                $ 899 "vr2_p3_up≔contact_fun(p[0,0,0,0,0,0],[0,1,0],20000,20,20)"
                global vr2_p3_up=contact_fun(p[0,0,0,0,0,0],[0,1,0],20000,20,20)
                $ 900 "direction(p[0,0,0,0,0,0],[0,-1,0],30,120,160)"
                direction(p[0,0,0,0,0,0],[0,-1,0],30,120,160)
                $ 901 "direction(p[0,0,0,0,0,0],[-1,0,0],20,120,160)"
                direction(p[0,0,0,0,0,0],[-1,0,0],20,120,160)
              end
              $ 902 "A_Touch_p[A_sel_v+9]=touch_4point(vr2_p1_up,vr2_p2_up,vr2_p3_up)"
              A_Touch_p[A_sel_v+9]=touch_4point(vr2_p1_up,vr2_p2_up,vr2_p3_up)
              $ 903 "A_Touch_p[A_sel_v+9]=ori_pose(A_Touch_p[A_sel_v+9],A_Touch_p[A_sel_v])"
              A_Touch_p[A_sel_v+9]=ori_pose(A_Touch_p[A_sel_v+9],A_Touch_p[A_sel_v])
            else:
              $ 904 "Else" "noBreak"
              $ 905 "If A_Touch_p[A_VR1]≟p[0,0,0,0,0,0]"
              if (A_Touch_p[A_VR1] == p[0,0,0,0,0,0]):
                $ 906 "Call MoveandTouchFun_3f"
                MoveandTouchFun_3f()
                $ 907 "touch_tmp≔A_Touch_p[A_sel_v]"
                global touch_tmp=A_Touch_p[A_sel_v]
                $ 908 "If A_Prepos_l[A_HOR_MR]≟p[0,0,0,0,0,0]"
                if (A_Prepos_l[A_HOR_MR] == p[0,0,0,0,0,0]):
                  $ 909 "direction(p[0,0,0,0,0,0],[-1,1,0],8,120,160)"
                  direction(p[0,0,0,0,0,0],[-1,1,0],8,120,160)
                  $ 910 "AAgcp≔get_actual_tcp_pose()"
                  global AAgcp= get_actual_tcp_pose ()
                  $ 911 "AAgangle≔up_right"
                  global AAgangle=p[.445203173045, -.406687378356, -.031125942276, 2.308490741423, -1.066468937023, 1.322151316133]
                  $ 912 "AAgtp≔p[AAgcp[0],AAgcp[1],AAgcp[2],AAgangle[3],AAgangle[4],AAgangle[5]]"
                  global AAgtp=p[AAgcp[0],AAgcp[1],AAgcp[2],AAgangle[3],AAgangle[4],AAgangle[5]]
                  $ 913 "MoveL"
                  $ 914 "AAgtp" "breakAfter"
                  movel(pose_trans(Base, AAgtp), a=0.08, v=0.08)
                  $ 916 "for_z_VLR2≔contact_fun(p[0,0,0,0,0,0],[0,0,-1],20000,20,20)"
                  global for_z_VLR2=contact_fun(p[0,0,0,0,0,0],[0,0,-1],20000,20,20)
                  $ 917 "touch_tmp[2]=for_z_VLR2[2]"
                  touch_tmp[2]=for_z_VLR2[2]
                end
                $ 918 "A_Touch_p[A_sel_v]=touch_tmp"
                A_Touch_p[A_sel_v]=touch_tmp
                $ 919 "for_cal_y_wel≔A_Touch_p[A_sel_v]"
                global for_cal_y_wel=A_Touch_p[A_sel_v]
                $ 920 "for_cal_x_wel≔A_Touch_p[A_sel_v]"
                global for_cal_x_wel=A_Touch_p[A_sel_v]
              else:
                $ 921 "Else" "noBreak"
                $ 922 "If A_Prepos_l[A_HOR_MR]≟p[0,0,0,0,0,0]"
                if (A_Prepos_l[A_HOR_MR] == p[0,0,0,0,0,0]):
                  $ 923 "Call MoveFun"
                  MoveFun()
                  $ 924 "for_cal_y_wel≔contact_fun(p[0,0,0,0,0,0],[1,0,0],20000,20,20)"
                  global for_cal_y_wel=contact_fun(p[0,0,0,0,0,0],[1,0,0],20000,20,20)
                  $ 925 "direction(p[0,0,0,0,0,0],[-1,0,0],40,120,160)"
                  direction(p[0,0,0,0,0,0],[-1,0,0],40,120,160)
                  $ 926 "direction(p[0,0,0,0,0,0],[0,-1,0],60,120,160)"
                  direction(p[0,0,0,0,0,0],[0,-1,0],60,120,160)
                  $ 927 "var_2≔contact_fun(p[0,0,0,0,0,0],[1,0,0],20000,20,20)"
                  global var_2=contact_fun(p[0,0,0,0,0,0],[1,0,0],20000,20,20)
                  $ 928 "direction(p[0,0,0,0,0,0],[-1,0,0],5,120,160)"
                  direction(p[0,0,0,0,0,0],[-1,0,0],5,120,160)
                  $ 929 "direction(p[0,0,0,0,0,0],[0,1,0],60,120,160)"
                  direction(p[0,0,0,0,0,0],[0,1,0],60,120,160)
                  $ 930 "direction(p[0,0,0,0,0,0],[1,0,0],10,120,160)"
                  direction(p[0,0,0,0,0,0],[1,0,0],10,120,160)
                  $ 931 "for_cal_x_wel≔contact_fun(p[0,0,0,0,0,0],[0,-1,0],20000,20,20)"
                  global for_cal_x_wel=contact_fun(p[0,0,0,0,0,0],[0,-1,0],20000,20,20)
                  $ 932 "direction(p[0,0,0,0,0,0],[0,1,0],20,120,160)"
                  direction(p[0,0,0,0,0,0],[0,1,0],20,120,160)
                  $ 933 "AAgcp≔get_actual_tcp_pose()"
                  global AAgcp= get_actual_tcp_pose ()
                  $ 934 "AAgangle≔up_right"
                  global AAgangle=p[.445203173045, -.406687378356, -.031125942276, 2.308490741423, -1.066468937023, 1.322151316133]
                  $ 935 "AAgtp≔p[AAgcp[0],AAgcp[1],AAgcp[2],AAgangle[3],AAgangle[4],AAgangle[5]]"
                  global AAgtp=p[AAgcp[0],AAgcp[1],AAgcp[2],AAgangle[3],AAgangle[4],AAgangle[5]]
                  $ 936 "MoveL"
                  $ 937 "AAgtp" "breakAfter"
                  movel(pose_trans(Base, AAgtp), a=0.1, v=0.1)
                  $ 939 "for_z_VLR2≔contact_fun(p[0,0,0,0,0,0],[0,0,-1],20000,20,20)"
                  global for_z_VLR2=contact_fun(p[0,0,0,0,0,0],[0,0,-1],20000,20,20)
                  $ 940 "direction(p[0,0,0,0,0,0],[0,0,1],20,120,160)"
                  direction(p[0,0,0,0,0,0],[0,0,1],20,120,160)
                  $ 941 "direction(p[0,0,0,0,0,0],[-1,0,0],20,120,160)"
                  direction(p[0,0,0,0,0,0],[-1,0,0],20,120,160)
                end
                $ 942 "for_cal_rot≔A_Touch_p[A_VR1]"
                global for_cal_rot=A_Touch_p[A_VR1]
                $ 944 "touch_tmp=p[for_cal_y_wel[0],for_cal_x_wel[1],for_cal_x_wel[2],for_cal_rot[3],for_cal_rot[4],for_cal_rot[5]]"
                touch_tmp=p[for_cal_y_wel[0],for_cal_x_wel[1],for_cal_x_wel[2],for_cal_rot[3],for_cal_rot[4],for_cal_rot[5]]
                $ 945 "If Scallup_check≟ False "
                if (Scallup_check ==   False  ):
                  $ 946 "touch_tmp≔pose_trans(touch_tmp,p[-(Touch_dis)/1000,0,0,0,0,0])"
                  global touch_tmp= pose_trans (touch_tmp,p[-(Touch_dis)/1000,0,0,0,0,0])
                else:
                  $ 947 "Else" "noBreak"
                  $ 948 "Scallup_check≔ False "
                  global Scallup_check=  False
                end
                $ 949 "A_Touch_p[A_sel_v]=touch_tmp"
                A_Touch_p[A_sel_v]=touch_tmp
                $ 950 "write_welder(4, False )"
                write_welder(4,  False  )
              end
            end
            $ 951 "b2_par_cd≔0"
            global b2_par_cd=0
            $ 952 "homeing()"
            homeing()
          else:
            $ 953 "Else" "noBreak"
            $ 954 "homeing()"
            homeing()
          end
          $ 955 "write_welder(4,False)"
          write_welder(4,False)
          $ 1012 "Touch After Offset"
          $ 1013 "touch_after_offset"
          $ 1014 "HOR"
          $ 1015 "If A_Prepos_l[A_HOR]≠p[0,0,0,0,0,0]"
          if (A_Prepos_l[A_HOR] != p[0,0,0,0,0,0]):
            $ 1016 "If b1_cell_info_L≟A or b1_cell_info_L≟C or b1_cell_info_L≟c"
            if (b1_cell_info_L == A  or  b1_cell_info_L == C  or  b1_cell_info_L == c):
              $ 1017 "If for_x_HOR≟p[0,0,0,0,0,0] and A_Touch_p[A_VL1]≠p[0,0,0,0,0,0]"
              if (for_x_HOR == p[0,0,0,0,0,0]  and  A_Touch_p[A_VL1] != p[0,0,0,0,0,0]):
                $ 1018 "for_x_HOR≔A_Touch_p[A_VL1]"
                global for_x_HOR=A_Touch_p[A_VL1]
              end
              $ 1019 "If for_x_HOR≠p[0,0,0,0,0,0]"
              if (for_x_HOR != p[0,0,0,0,0,0]):
                $ 1020 "x_diff≔get_feature_pose(for_x_HOR,A_Touch_p[A_HOR])"
                global x_diff=get_feature_pose(for_x_HOR,A_Touch_p[A_HOR])
                $ 1021 "A_Touch_p[A_HOR]=pose_trans(A_Touch_p[A_HOR], p[x_diff[0],0,0,0,0,0])"
                A_Touch_p[A_HOR]= pose_trans (A_Touch_p[A_HOR], p[x_diff[0],0,0,0,0,0])
                $ 1022 "If b1_cell_info_L≟B or b1_cell_info_L≟D or b1_cell_info_L≟d or b1_cell_info_L≟E or b1_cell_info_L≟e"
                if (b1_cell_info_L == B  or  b1_cell_info_L == D  or  b1_cell_info_L == d  or  b1_cell_info_L == E  or  b1_cell_info_L == e):
                  $ 1023 "A_Touch_p[A_HOR]=pose_trans(A_Touch_p[A_HOR], p[hor_l_scallup/1000,0,0,0,0,0])"
                  A_Touch_p[A_HOR]= pose_trans (A_Touch_p[A_HOR], p[hor_l_scallup/1000,0,0,0,0,0])
                end
              end
            end
            $ 1024 "A_Touch_p[A_HOR]=pose_trans(A_Touch_p[A_HOR], p[offset_2f_begin/1000,0,0,0,0,0])"
            A_Touch_p[A_HOR]= pose_trans (A_Touch_p[A_HOR], p[offset_2f_begin/1000,0,0,0,0,0])
          end
          $ 1025 "VL1"
          $ 1026 "If A_Prepos_l[A_VL1]≠p[0,0,0,0,0,0]"
          if (A_Prepos_l[A_VL1] != p[0,0,0,0,0,0]):
            $ 1027 "If b1_cell_info_L≟A or b1_cell_info_L≟C or b1_cell_info_L≟c"
            if (b1_cell_info_L == A  or  b1_cell_info_L == C  or  b1_cell_info_L == c):
              $ 1028 "'3f only does not apply offset'"
              # '3f only does not apply offset'
              $ 1029 "If for_z_VL1≟p[0,0,0,0,0,0] and A_Touch_p[A_HOR]≠p[0,0,0,0,0,0]"
              if (for_z_VL1 == p[0,0,0,0,0,0]  and  A_Touch_p[A_HOR] != p[0,0,0,0,0,0]):
                $ 1030 "for_z_VL1≔A_Touch_p[A_HOR]"
                global for_z_VL1=A_Touch_p[A_HOR]
              end
              $ 1031 "Comment"
              # Comment
              $ 1032 "If for_z_VL1≠p[0,0,0,0,0,0]"
              if (for_z_VL1 != p[0,0,0,0,0,0]):
                $ 1033 "z_diff≔get_feature_pose(for_z_VL1,A_Touch_p[A_VL1])"
                global z_diff=get_feature_pose(for_z_VL1,A_Touch_p[A_VL1])
                $ 1034 "A_Touch_p[A_VL1]=pose_trans(A_Touch_p[A_VL1], p[z_diff[0],0,0,0,0,0])"
                A_Touch_p[A_VL1]= pose_trans (A_Touch_p[A_VL1], p[z_diff[0],0,0,0,0,0])
              end
              $ 1035 "If b1_cell_info_L≟B or b1_cell_info_L≟D or b1_cell_info_L≟d or b1_cell_info_L≟E or b1_cell_info_L≟e"
              if (b1_cell_info_L == B  or  b1_cell_info_L == D  or  b1_cell_info_L == d  or  b1_cell_info_L == E  or  b1_cell_info_L == e):
                $ 1036 "A_Touch_p[A_VL1]=pose_trans(A_Touch_p[A_VL1], p[vert_scallup_l/1000,0,0,0,0,0])"
                A_Touch_p[A_VL1]= pose_trans (A_Touch_p[A_VL1], p[vert_scallup_l/1000,0,0,0,0,0])
              end
            end
            $ 1038 "A_Touch_p[A_VL1]=pose_trans(A_Touch_p[A_VL1], p[offset_3f_begin/1000,0,0,0,0,0])"
            A_Touch_p[A_VL1]= pose_trans (A_Touch_p[A_VL1], p[offset_3f_begin/1000,0,0,0,0,0])
          end
          $ 1039 "VL2"
          $ 1040 "If A_Prepos_l[A_VL2]≠p[0,0,0,0,0,0]"
          if (A_Prepos_l[A_VL2] != p[0,0,0,0,0,0]):
            $ 1041 "If b1_cell_info_L≟A or b1_cell_info_L≟C or b1_cell_info_L≟c or b1_cell_info_L≟D or b1_cell_info_L≟d or b1_cell_info_L≟E"
            if (b1_cell_info_L == A  or  b1_cell_info_L == C  or  b1_cell_info_L == c  or  b1_cell_info_L == D  or  b1_cell_info_L == d  or  b1_cell_info_L == E):
              $ 1042 "'3f only does not apply offset'"
              # '3f only does not apply offset'
              $ 1043 "If for_z_VLR2≟p[0,0,0,0,0,0] and A_Touch_p[A_HOR_ML]≠p[0,0,0,0,0,0]"
              if (for_z_VLR2 == p[0,0,0,0,0,0]  and  A_Touch_p[A_HOR_ML] != p[0,0,0,0,0,0]):
                $ 1044 "for_z_VLR2≔A_Touch_p[A_HOR_ML]"
                global for_z_VLR2=A_Touch_p[A_HOR_ML]
              end
              $ 1045 "Comment"
              # Comment
              $ 1046 "If for_z_VLR2≠p[0,0,0,0,0,0]"
              if (for_z_VLR2 != p[0,0,0,0,0,0]):
                $ 1047 "z_diff≔get_feature_pose(for_z_VLR2,A_Touch_p[A_VL2])"
                global z_diff=get_feature_pose(for_z_VLR2,A_Touch_p[A_VL2])
                $ 1048 "A_Touch_p[A_VL2]=pose_trans(A_Touch_p[A_VL2], p[z_diff[0],0,0,0,0,0])"
                A_Touch_p[A_VL2]= pose_trans (A_Touch_p[A_VL2], p[z_diff[0],0,0,0,0,0])
              end
              $ 1049 "If b1_cell_info_L≟E or b1_cell_info_L≟e"
              if (b1_cell_info_L == E  or  b1_cell_info_L == e):
                $ 1050 "A_Touch_p[A_VL2]=pose_trans(A_Touch_p[A_VL2], p[vert_scallup_l/1000,0,0,0,0,0])"
                A_Touch_p[A_VL2]= pose_trans (A_Touch_p[A_VL2], p[vert_scallup_l/1000,0,0,0,0,0])
              end
            end
            $ 1051 "A_Touch_p[A_VL2]=pose_trans(A_Touch_p[A_VL2], p[offset_3f_begin/1000,0,0,0,0,0])"
            A_Touch_p[A_VL2]= pose_trans (A_Touch_p[A_VL2], p[offset_3f_begin/1000,0,0,0,0,0])
          end
          $ 1052 "HOR_R"
          $ 1053 "If A_Prepos_l[A_HOR_R]≠p[0,0,0,0,0,0]"
          if (A_Prepos_l[A_HOR_R] != p[0,0,0,0,0,0]):
            $ 1054 "If b1_cell_info_R≟A or b1_cell_info_R≟C or b1_cell_info_R≟c"
            if (b1_cell_info_R == A  or  b1_cell_info_R == C  or  b1_cell_info_R == c):
              $ 1055 "If for_x_HOR_R≟p[0,0,0,0,0,0] and A_Touch_p[A_VR1]≠p[0,0,0,0,0,0]"
              if (for_x_HOR_R == p[0,0,0,0,0,0]  and  A_Touch_p[A_VR1] != p[0,0,0,0,0,0]):
                $ 1056 "for_x_HOR_R≔A_Touch_p[A_VR1]"
                global for_x_HOR_R=A_Touch_p[A_VR1]
              end
              $ 1057 "If for_x_HOR≠p[0,0,0,0,0,0]"
              if (for_x_HOR != p[0,0,0,0,0,0]):
                $ 1058 "x_diff≔get_feature_pose(for_x_HOR_R,A_Touch_p[A_HOR_R])"
                global x_diff=get_feature_pose(for_x_HOR_R,A_Touch_p[A_HOR_R])
                $ 1059 "A_Touch_p[A_HOR_R]=pose_trans(A_Touch_p[A_HOR_R], p[x_diff[0],0,0,0,0,0])"
                A_Touch_p[A_HOR_R]= pose_trans (A_Touch_p[A_HOR_R], p[x_diff[0],0,0,0,0,0])
                $ 1060 "If b1_cell_info_R≟B or b1_cell_info_R≟D or b1_cell_info_R≟d or b1_cell_info_R≟E or b1_cell_info_R≟e"
                if (b1_cell_info_R == B  or  b1_cell_info_R == D  or  b1_cell_info_R == d  or  b1_cell_info_R == E  or  b1_cell_info_R == e):
                  $ 1061 "A_Touch_p[A_HOR_R]=pose_trans(A_Touch_p[A_HOR_R], p[-hor_r_scallup/1000,0,0,0,0,0])"
                  A_Touch_p[A_HOR_R]= pose_trans (A_Touch_p[A_HOR_R], p[-hor_r_scallup/1000,0,0,0,0,0])
                end
              end
            end
            $ 1062 "A_Touch_p[A_HOR_R]=pose_trans(A_Touch_p[A_HOR_R], p[-offset_2f_begin/1000,0,0,0,0,0])"
            A_Touch_p[A_HOR_R]= pose_trans (A_Touch_p[A_HOR_R], p[-offset_2f_begin/1000,0,0,0,0,0])
          end
          $ 1063 "VR1"
          $ 1064 "If A_Prepos_l[A_VR1]≠p[0,0,0,0,0,0]"
          if (A_Prepos_l[A_VR1] != p[0,0,0,0,0,0]):
            $ 1065 "If b1_cell_info_R≟A or b1_cell_info_R≟C or b1_cell_info_R≟c"
            if (b1_cell_info_R == A  or  b1_cell_info_R == C  or  b1_cell_info_R == c):
              $ 1066 "If for_z_VR1≟p[0,0,0,0,0,0] and A_Touch_p[A_HOR_R]≠p[0,0,0,0,0,0]"
              if (for_z_VR1 == p[0,0,0,0,0,0]  and  A_Touch_p[A_HOR_R] != p[0,0,0,0,0,0]):
                $ 1067 "for_z_VR1≔A_Touch_p[A_HOR_R]"
                global for_z_VR1=A_Touch_p[A_HOR_R]
              end
              $ 1068 "If for_z_VR1≠p[0,0,0,0,0,0]"
              if (for_z_VR1 != p[0,0,0,0,0,0]):
                $ 1069 "z_diff≔get_feature_pose(for_z_VR1,A_Touch_p[A_VR1])"
                global z_diff=get_feature_pose(for_z_VR1,A_Touch_p[A_VR1])
                $ 1070 "A_Touch_p[A_VR1]=pose_trans(A_Touch_p[A_VR1], p[z_diff[0],0,0,0,0,0])"
                A_Touch_p[A_VR1]= pose_trans (A_Touch_p[A_VR1], p[z_diff[0],0,0,0,0,0])
              end
              $ 1071 "If b1_cell_info_R≟B or b1_cell_info_R≟D or b1_cell_info_R≟d or b1_cell_info_R≟E or b1_cell_info_R≟e"
              if (b1_cell_info_R == B  or  b1_cell_info_R == D  or  b1_cell_info_R == d  or  b1_cell_info_R == E  or  b1_cell_info_R == e):
                $ 1072 "A_Touch_p[A_VR1]=pose_trans(A_Touch_p[A_VR1], p[vert_scallup_r/1000,0,0,0,0,0])"
                A_Touch_p[A_VR1]= pose_trans (A_Touch_p[A_VR1], p[vert_scallup_r/1000,0,0,0,0,0])
              end
            end
            $ 1074 "A_Touch_p[A_VR1]=pose_trans(A_Touch_p[A_VR1], p[offset_3f_begin/1000,0,0,0,0,0])"
            A_Touch_p[A_VR1]= pose_trans (A_Touch_p[A_VR1], p[offset_3f_begin/1000,0,0,0,0,0])
          end
          $ 1075 "VR2"
          $ 1076 "If A_Prepos_l[A_VR2]≠p[0,0,0,0,0,0]"
          if (A_Prepos_l[A_VR2] != p[0,0,0,0,0,0]):
            $ 1077 "If b1_cell_info_R≟A or b1_cell_info_R≟C or b1_cell_info_R≟c or b1_cell_info_R≟D or b1_cell_info_R≟d or b1_cell_info_R≟E"
            if (b1_cell_info_R == A  or  b1_cell_info_R == C  or  b1_cell_info_R == c  or  b1_cell_info_R == D  or  b1_cell_info_R == d  or  b1_cell_info_R == E):
              $ 1078 "'3f only does not apply offset'"
              # '3f only does not apply offset'
              $ 1079 "If for_z_VLR2≟p[0,0,0,0,0,0] and A_Touch_p[A_HOR_MR]≠p[0,0,0,0,0,0]"
              if (for_z_VLR2 == p[0,0,0,0,0,0]  and  A_Touch_p[A_HOR_MR] != p[0,0,0,0,0,0]):
                $ 1080 "for_z_VLR2≔A_Touch_p[A_HOR_MR]"
                global for_z_VLR2=A_Touch_p[A_HOR_MR]
              end
              $ 1081 "Comment"
              # Comment
              $ 1082 "If for_z_VLR2≠p[0,0,0,0,0,0]"
              if (for_z_VLR2 != p[0,0,0,0,0,0]):
                $ 1083 "z_diff≔get_feature_pose(for_z_VLR2,A_Touch_p[A_VR2])"
                global z_diff=get_feature_pose(for_z_VLR2,A_Touch_p[A_VR2])
                $ 1084 "A_Touch_p[A_VR2]=pose_trans(A_Touch_p[A_VR2], p[z_diff[0],0,0,0,0,0])"
                A_Touch_p[A_VR2]= pose_trans (A_Touch_p[A_VR2], p[z_diff[0],0,0,0,0,0])
              end
              $ 1085 "If b1_cell_info_R≟E or b1_cell_info_R≟e"
              if (b1_cell_info_R == E  or  b1_cell_info_R == e):
                $ 1086 "A_Touch_p[A_VR2]=pose_trans(A_Touch_p[A_VR2], p[vert_scallup_r/1000,0,0,0,0,0])"
                A_Touch_p[A_VR2]= pose_trans (A_Touch_p[A_VR2], p[vert_scallup_r/1000,0,0,0,0,0])
              end
            end
            $ 1087 "A_Touch_p[A_VR2]=pose_trans(A_Touch_p[A_VR2], p[offset_3f_begin/1000,0,0,0,0,0])"
            A_Touch_p[A_VR2]= pose_trans (A_Touch_p[A_VR2], p[offset_3f_begin/1000,0,0,0,0,0])
          end
          $ 1088 "HOR_ML"
          $ 1089 "If A_Prepos_l[A_HOR_ML]≠p[0,0,0,0,0,0]"
          if (A_Prepos_l[A_HOR_ML] != p[0,0,0,0,0,0]):
            $ 1090 "A_Touch_p[A_HOR_M]=A_Touch_p[A_HOR_ML]"
            A_Touch_p[A_HOR_M]=A_Touch_p[A_HOR_ML]
            $ 1091 "x_welding_axis≔get_feature_pose(for_cal_x_wel,A_Touch_p[A_HOR_ML])"
            global x_welding_axis=get_feature_pose(for_cal_x_wel,A_Touch_p[A_HOR_ML])
            $ 1092 "A_Touch_p[A_HOR_M]=pose_trans(A_Touch_p[A_HOR_ML], p[x_welding_axis[0],0,0,0,0,0])"
            A_Touch_p[A_HOR_M]= pose_trans (A_Touch_p[A_HOR_ML], p[x_welding_axis[0],0,0,0,0,0])
            $ 1093 "A_Touch_p[A_HOR_M]=put_pose(A_Touch_p[A_HOR_M],0,for_cal_y_wel[0])"
            A_Touch_p[A_HOR_M]=put_pose(A_Touch_p[A_HOR_M],0,for_cal_y_wel[0])
            $ 1094 "A_Touch_p[A_HOR_M]=pose_trans(A_Touch_p[A_HOR_M], p[10/1000,0,0,0,0,0])"
            A_Touch_p[A_HOR_M]= pose_trans (A_Touch_p[A_HOR_M], p[10/1000,0,0,0,0,0])
            $ 1095 "If b1_cell_info_L≟C or b1_cell_info_L≟D"
            if (b1_cell_info_L == C  or  b1_cell_info_L == D):
              $ 1097 "x_welding_axis≔get_feature_pose(for_cal_x_wel,A_Touch_p[A_HOR_ML])"
              global x_welding_axis=get_feature_pose(for_cal_x_wel,A_Touch_p[A_HOR_ML])
              $ 1098 "A_Touch_p[A_HOR_ML]=pose_trans(A_Touch_p[A_HOR_ML],p[x_welding_axis[0],0,0,0,0,0])"
              A_Touch_p[A_HOR_ML]= pose_trans (A_Touch_p[A_HOR_ML],p[x_welding_axis[0],0,0,0,0,0])
              $ 1099 "A_Touch_p[A_HOR_ML]=pose_trans(A_Touch_p[A_HOR_ML],p[0/1000,0,0,0,0,0])"
              A_Touch_p[A_HOR_ML]= pose_trans (A_Touch_p[A_HOR_ML],p[0/1000,0,0,0,0,0])
            end
          end
          $ 1100 "HOR_MR"
          $ 1101 "If A_Prepos_l[A_HOR_MR]≠p[0,0,0,0,0,0]"
          if (A_Prepos_l[A_HOR_MR] != p[0,0,0,0,0,0]):
            $ 1103 "A_Touch_p[A_HOR_M]=A_Touch_p[A_HOR_MR]"
            A_Touch_p[A_HOR_M]=A_Touch_p[A_HOR_MR]
            $ 1104 "x_welding_axis≔get_feature_pose(for_cal_x_wel,A_Touch_p[A_HOR_MR])"
            global x_welding_axis=get_feature_pose(for_cal_x_wel,A_Touch_p[A_HOR_MR])
            $ 1105 "A_Touch_p[A_HOR_M]=pose_trans(A_Touch_p[A_HOR_M], p[x_welding_axis[0],0,0,0,0,0])"
            A_Touch_p[A_HOR_M]= pose_trans (A_Touch_p[A_HOR_M], p[x_welding_axis[0],0,0,0,0,0])
            $ 1106 "A_Touch_p[A_HOR_M]=put_pose(A_Touch_p[A_HOR_M],0,for_cal_y_wel[0])"
            A_Touch_p[A_HOR_M]=put_pose(A_Touch_p[A_HOR_M],0,for_cal_y_wel[0])
            $ 1107 "A_Touch_p[A_HOR_M]=pose_trans(A_Touch_p[A_HOR_M], p[-10/1000,0,0,0,0,0])"
            A_Touch_p[A_HOR_M]= pose_trans (A_Touch_p[A_HOR_M], p[-10/1000,0,0,0,0,0])
            $ 1108 "If b1_cell_info_R≟C or b1_cell_info_R≟D"
            if (b1_cell_info_R == C  or  b1_cell_info_R == D):
              $ 1110 "x_welding_axis≔get_feature_pose(for_cal_x_wel,A_Touch_p[A_HOR_MR])"
              global x_welding_axis=get_feature_pose(for_cal_x_wel,A_Touch_p[A_HOR_MR])
              $ 1111 "A_Touch_p[A_HOR_MR]=pose_trans(A_Touch_p[A_HOR_MR],p[x_welding_axis[0],0,0,0,0,0])"
              A_Touch_p[A_HOR_MR]= pose_trans (A_Touch_p[A_HOR_MR],p[x_welding_axis[0],0,0,0,0,0])
              $ 1112 "A_Touch_p[A_HOR_MR]=pose_trans(A_Touch_p[A_HOR_MR],p[-0/1000,0,0,0,0,0])"
              A_Touch_p[A_HOR_MR]= pose_trans (A_Touch_p[A_HOR_MR],p[-0/1000,0,0,0,0,0])
            end
          end
          $ 1113 "'Touch Remember On/OFF'"
          # 'Touch Remember On/OFF'
          $ 1114 "write_port_register(180,1)"
          write_port_register(180,1)
        else:
          $ 1115 "Else" "noBreak"
          $ 1116 "Ignore Touch and check error"
          $ 1117 "Auto_cur_cell≔0"
          global Auto_cur_cell=0
          $ 1118 "Loop Auto_cur_cell<Auto_total_cell"
          while (Auto_cur_cell<Auto_total_cell):
            $ 1119 "A_sel_v≔Auto_W_num[Auto_cur_cell]"
            global A_sel_v=Auto_W_num[Auto_cur_cell]
            $ 1120 "If A_sel_v<A_HOR_2path"
            if (A_sel_v<A_HOR_2path):
              $ 1121 "If A_Touch_p[A_sel_v]≟p[0,0,0,0,0,0]"
              if (A_Touch_p[A_sel_v] == p[0,0,0,0,0,0]):
                $ 1122 "write_port_register(142,120)"
                write_port_register(142,120)
                $ 1123 "Halt"
                halt
              end
            end
            $ 1124 "Auto_cur_cell≔Auto_cur_cell+1"
            global Auto_cur_cell=Auto_cur_cell+1
          end
          $ 1125 "Auto_cur_cell≔0"
          global Auto_cur_cell=0
        end
        $ 1126 "welding"
        $ 1127 "weldings"
        $ 1128 "Auto_cur_cell≔read_port_register(138)"
        global Auto_cur_cell= read_port_register (138)
        $ 1129 "time_cal_trig≔ True "
        global time_cal_trig=  True
        $ 1130 "Loop Auto_cur_cell<Auto_total_cell"
        while (Auto_cur_cell<Auto_total_cell):
          $ 1131 "write_port_register(138,Auto_cur_cell)"
          write_port_register(138,Auto_cur_cell)
          $ 1132 "running_trig≔ True "
          global running_trig=  True
          $ 1133 "'[2F_AB - 30] , [2F_CD_LEFT - 100] , [2F_CD_RIGHT - 150] , [3F - ELSE]'"
          # '[2F_AB - 30] , [2F_CD_LEFT - 100] , [2F_CD_RIGHT - 150] , [3F - ELSE]'
          $ 1134 "If Auto_W_num[Auto_cur_cell]≥100 and Auto_W_num[Auto_cur_cell]≤149"
          if (Auto_W_num[Auto_cur_cell] >= 100  and  Auto_W_num[Auto_cur_cell] <= 149):
            $ 1135 "'2F CD LEFT'"
            # '2F CD LEFT'
            $ 1136 "A_sel_v≔A_HOR"
            global A_sel_v=A_HOR
            $ 1137 "A_sel_v_end≔A_HOR_ML"
            global A_sel_v_end=A_HOR_ML
            $ 1138 "A_sel_v2≔A_HOR_M"
            global A_sel_v2=A_HOR_M
            $ 1139 "A_sel_v_end2≔A_HOR_R"
            global A_sel_v_end2=A_HOR_R
            $ 1140 "If floor(Auto_W_num[Auto_cur_cell]/10)≟10"
            if (floor(Auto_W_num[Auto_cur_cell]/10) == 10):
              $ 1141 "current_path≔1"
              global current_path=1
              $ 1142 "multi_path≔1"
              global multi_path=1
            else:
              $ 1143 "ElseIf floor(Auto_W_num[Auto_cur_cell]/10)≟11"
              if (floor(Auto_W_num[Auto_cur_cell]/10) == 11):
                $ 1144 "current_path≔2"
                global current_path=2
                $ 1145 "multi_path≔2"
                global multi_path=2
              else:
                $ 1146 "ElseIf floor(Auto_W_num[Auto_cur_cell]/10)≟12"
                if (floor(Auto_W_num[Auto_cur_cell]/10) == 12):
                  $ 1147 "current_path≔3"
                  global current_path=3
                  $ 1148 "multi_path≔3"
                  global multi_path=3
                else:
                  $ 1149 "ElseIf floor(Auto_W_num[Auto_cur_cell]/10)≟13"
                  if (floor(Auto_W_num[Auto_cur_cell]/10) == 13):
                    $ 1150 "current_path≔4"
                    global current_path=4
                    $ 1151 "multi_path≔4"
                    global multi_path=4
                  end
                end
              end
            end
            $ 1152 "current_2f≔current_2f+1"
            global current_2f=current_2f+1
            $ 1153 "CD_MLR≔ True "
            global CD_MLR=  True
            $ 1154 "write_port_register(135,A_HOR)"
            write_port_register(135,A_HOR)
            $ 1155 "write_port_register(136,current_2f)"
            write_port_register(136,current_2f)
            $ 1156 "If simulation_mode"
            if (simulation_mode):
              $ 1157 "Call welding_parameter_sim"
              welding_parameter_sim()
            else:
              $ 1158 "Else" "noBreak"
              $ 1159 "Call welding_parameter_init"
              welding_parameter_init()
            end
            $ 1160 "wv_direction≔1"
            global wv_direction=1
            $ 1161 "If Auto_W_num[Auto_cur_cell]%10≟4"
            if (Auto_W_num[Auto_cur_cell]%10 == 4):
              $ 1162 "A_sel_v≔A_HOR_R"
              global A_sel_v=A_HOR_R
              $ 1163 "Call MoveFun"
              MoveFun()
              $ 1164 "A_sel_v≔A_HOR"
              global A_sel_v=A_HOR
            else:
              $ 1165 "ElseIf Auto_W_num[Auto_cur_cell]%10≟0 or Auto_W_num[Auto_cur_cell]%10≟1 or Auto_W_num[Auto_cur_cell]%10≟2"
              if (Auto_W_num[Auto_cur_cell]%10 == 0  or  Auto_W_num[Auto_cur_cell]%10 == 1  or  Auto_W_num[Auto_cur_cell]%10 == 2):
                $ 1166 "Call MoveFun"
                MoveFun()
              end
            end
            $ 1167 "Call weav_welding_2f_CD"
            weav_welding_2f_CD()
          else:
            $ 1168 "ElseIf Auto_W_num[Auto_cur_cell]≥150 and Auto_W_num[Auto_cur_cell]≤189"
            if (Auto_W_num[Auto_cur_cell] >= 150  and  Auto_W_num[Auto_cur_cell] <= 189):
              $ 1169 "'2F CD RIGHT'"
              # '2F CD RIGHT'
              $ 1170 "A_sel_v≔A_HOR_R"
              global A_sel_v=A_HOR_R
              $ 1171 "A_sel_v_end≔A_HOR_MR"
              global A_sel_v_end=A_HOR_MR
              $ 1172 "A_sel_v2≔A_HOR_M"
              global A_sel_v2=A_HOR_M
              $ 1173 "A_sel_v_end2≔A_HOR"
              global A_sel_v_end2=A_HOR
              $ 1174 "If floor(Auto_W_num[Auto_cur_cell]/10)≟15"
              if (floor(Auto_W_num[Auto_cur_cell]/10) == 15):
                $ 1175 "current_path≔1"
                global current_path=1
                $ 1176 "multi_path≔1"
                global multi_path=1
              else:
                $ 1177 "ElseIf floor(Auto_W_num[Auto_cur_cell]/10)≟16"
                if (floor(Auto_W_num[Auto_cur_cell]/10) == 16):
                  $ 1178 "current_path≔2"
                  global current_path=2
                  $ 1179 "multi_path≔2"
                  global multi_path=2
                else:
                  $ 1180 "ElseIf floor(Auto_W_num[Auto_cur_cell]/10)≟17"
                  if (floor(Auto_W_num[Auto_cur_cell]/10) == 17):
                    $ 1181 "current_path≔3"
                    global current_path=3
                    $ 1182 "multi_path≔3"
                    global multi_path=3
                  else:
                    $ 1183 "ElseIf floor(Auto_W_num[Auto_cur_cell]/10)≟18"
                    if (floor(Auto_W_num[Auto_cur_cell]/10) == 18):
                      $ 1184 "current_path≔4"
                      global current_path=4
                      $ 1185 "multi_path≔4"
                      global multi_path=4
                    end
                  end
                end
              end
              $ 1186 "current_2f≔current_2f+1"
              global current_2f=current_2f+1
              $ 1187 "CD_MLR≔ False "
              global CD_MLR=  False
              $ 1188 "write_port_register(135,A_HOR)"
              write_port_register(135,A_HOR)
              $ 1189 "write_port_register(136,current_2f)"
              write_port_register(136,current_2f)
              $ 1190 "If simulation_mode"
              if (simulation_mode):
                $ 1191 "Call welding_parameter_sim"
                welding_parameter_sim()
              else:
                $ 1192 "Else" "noBreak"
                $ 1193 "Call welding_parameter_init"
                welding_parameter_init()
              end
              $ 1194 "wv_direction≔-1"
              global wv_direction=-1
              $ 1195 "If Auto_W_num[Auto_cur_cell]%10≟4"
              if (Auto_W_num[Auto_cur_cell]%10 == 4):
                $ 1196 "A_sel_v≔A_HOR"
                global A_sel_v=A_HOR
                $ 1197 "Call MoveFun"
                MoveFun()
                $ 1198 "A_sel_v≔A_HOR_R"
                global A_sel_v=A_HOR_R
              else:
                $ 1199 "ElseIf Auto_W_num[Auto_cur_cell]%10≟0 or Auto_W_num[Auto_cur_cell]%10≟1 or Auto_W_num[Auto_cur_cell]%10≟2"
                if (Auto_W_num[Auto_cur_cell]%10 == 0  or  Auto_W_num[Auto_cur_cell]%10 == 1  or  Auto_W_num[Auto_cur_cell]%10 == 2):
                  $ 1200 "Call MoveFun"
                  MoveFun()
                end
              end
              $ 1201 "Call weav_welding_2f_CD"
              weav_welding_2f_CD()
            else:
              $ 1202 "ElseIf Auto_W_num[Auto_cur_cell]≥30 and Auto_W_num[Auto_cur_cell]≤65"
              if (Auto_W_num[Auto_cur_cell] >= 30  and  Auto_W_num[Auto_cur_cell] <= 65):
                $ 1203 "'2F'"
                # '2F'
                $ 1204 "A_sel_v≔A_HOR"
                global A_sel_v=A_HOR
                $ 1205 "A_sel_v_end≔A_HOR_R"
                global A_sel_v_end=A_HOR_R
                $ 1206 "If floor(Auto_W_num[Auto_cur_cell]/10)≟3"
                if (floor(Auto_W_num[Auto_cur_cell]/10) == 3):
                  $ 1207 "current_path≔1"
                  global current_path=1
                  $ 1208 "multi_path≔1"
                  global multi_path=1
                else:
                  $ 1209 "ElseIf floor(Auto_W_num[Auto_cur_cell]/10)≟4"
                  if (floor(Auto_W_num[Auto_cur_cell]/10) == 4):
                    $ 1210 "current_path≔2"
                    global current_path=2
                    $ 1211 "multi_path≔2"
                    global multi_path=2
                  else:
                    $ 1212 "ElseIf floor(Auto_W_num[Auto_cur_cell]/10)≟5"
                    if (floor(Auto_W_num[Auto_cur_cell]/10) == 5):
                      $ 1213 "current_path≔3"
                      global current_path=3
                      $ 1214 "multi_path≔3"
                      global multi_path=3
                    else:
                      $ 1215 "ElseIf floor(Auto_W_num[Auto_cur_cell]/10)≟6"
                      if (floor(Auto_W_num[Auto_cur_cell]/10) == 6):
                        $ 1216 "current_path≔4"
                        global current_path=4
                        $ 1217 "multi_path≔4"
                        global multi_path=4
                      end
                    end
                  end
                end
                $ 1218 "current_2f≔current_2f+1"
                global current_2f=current_2f+1
                $ 1219 "write_port_register(135,A_HOR)"
                write_port_register(135,A_HOR)
                $ 1220 "write_port_register(136,current_2f)"
                write_port_register(136,current_2f)
                $ 1221 "If simulation_mode"
                if (simulation_mode):
                  $ 1222 "Call welding_parameter_sim"
                  welding_parameter_sim()
                else:
                  $ 1223 "Else" "noBreak"
                  $ 1224 "Call welding_parameter_init"
                  welding_parameter_init()
                end
                $ 1225 "If Auto_W_num[Auto_cur_cell]%10≟2"
                if (Auto_W_num[Auto_cur_cell]%10 == 2):
                  $ 1226 "A_sel_v≔A_HOR_R"
                  global A_sel_v=A_HOR_R
                  $ 1227 "Call MoveFun"
                  MoveFun()
                  $ 1228 "A_sel_v≔A_HOR"
                  global A_sel_v=A_HOR
                else:
                  $ 1229 "Else" "noBreak"
                  $ 1230 "Call MoveFun"
                  MoveFun()
                end
                $ 1231 "Call weav_welding_2f"
                weav_welding_2f()
              else:
                $ 1232 "Else" "noBreak"
                $ 1233 "A_sel_v≔Auto_W_num[Auto_cur_cell]"
                global A_sel_v=Auto_W_num[Auto_cur_cell]
                $ 1234 "write_port_register(135,A_sel_v)"
                write_port_register(135,A_sel_v)
                $ 1235 "current_path≔1"
                global current_path=1
                $ 1236 "current_2f≔0"
                global current_2f=0
                $ 1237 "write_port_register(136,current_2f)"
                write_port_register(136,current_2f)
                $ 1238 "If simulation_mode"
                if (simulation_mode):
                  $ 1239 "Call welding_parameter_sim"
                  welding_parameter_sim()
                else:
                  $ 1240 "Else" "noBreak"
                  $ 1241 "Call welding_parameter_init"
                  welding_parameter_init()
                end
                $ 1242 "A_sel_v_end≔A_sel_v+9"
                global A_sel_v_end=A_sel_v+9
                $ 1243 "Call weav_welding_3f"
                weav_welding_3f()
              end
            end
          end
          $ 1244 "Call reset_weld_param"
          reset_weld_param()
          $ 1245 "next_before"
          $ 1246 "If get_move_trig≟1"
          if (get_move_trig == 1):
            $ 1247 "If get_next_number≠Auto_cur_cell"
            if (get_next_number != Auto_cur_cell):
              $ 1248 "Auto_cur_cell≔get_next_number"
              global Auto_cur_cell=get_next_number
            else:
              $ 1249 "Else" "noBreak"
              $ 1250 "Auto_cur_cell≔Auto_cur_cell+1"
              global Auto_cur_cell=Auto_cur_cell+1
            end
            $ 1251 "write_port_register(166,0)"
            write_port_register(166,0)
            $ 1252 "write_port_register(167,0)"
            write_port_register(167,0)
            $ 1253 "get_move_trig≔0"
            global get_move_trig=0
          else:
            $ 1254 "Else" "noBreak"
            $ 1255 "Auto_cur_cell≔Auto_cur_cell+1"
            global Auto_cur_cell=Auto_cur_cell+1
          end
        end
        $ 1256 "homeing()"
        homeing()
        $ 1257 "write_port_register(162,1)"
        write_port_register(162,1)
        $ 1258 "write_port_register(180,0)"
        write_port_register(180,0)
        thread_flag_305 = 1
      end
      if (a0_Job_Mode == 2):
        global thread_handler_305=run Thread_if_305()
        while (thread_flag_305 == 0):
          if not(a0_Job_Mode == 2):
            kill thread_handler_305
            thread_flag_305 = 2
          else:
            sync()
          end
        end
      else:
        thread_flag_305 = 2
      end
    end
    $ 1259 "Wait: 0.01"
    sleep(0.01)
    $ 1260 "after init auto"
    $ 1261 "If auto_on"
    if (auto_on):
      $ 1262 "write_port_register(202,0)"
      write_port_register(202,0)
      $ 1263 "timer_1: Stop"
      timer_1_is_counting = False
      $ 1264 "write_welder(0, False )"
      write_welder(0,  False  )
      $ 1265 "write_welder(4, False )"
      write_welder(4,  False  )
      $ 1266 "Call reset_weld_param"
      reset_weld_param()
      $ 1267 "multi_path≔1"
      global multi_path=1
      $ 1268 "auto_on≔ False "
      global auto_on=  False
      $ 1269 "current_2f≔0"
      global current_2f=0
      $ 1270 "get_center≔get_center_bak"
      global get_center=get_center_bak
      $ 1271 "vr2_p1≔p[0,0,0,0,0,0]"
      global vr2_p1=p[0,0,0,0,0,0]
      $ 1272 "welding_program≔ False "
      global welding_program=  False
      $ 1273 "start_num≔135"
      global start_num=135
      $ 1274 "Loop start_num<141"
      while (start_num<141):
        $ 1275 "write_port_register(start_num,0)"
        write_port_register(start_num,0)
        $ 1276 "start_num≔start_num+1"
        global start_num=start_num+1
      end
    end
  end
end
